PROGRAM MAIN
VAR_OUTPUT //globally readable, but only modifiable by MAIN
	outputBuffer : ARRAY[Surface.LEFT..Surface.RIGHT] OF Bundle;
	outputBufferPass, outputBufferFail : Bundle;
	numOutputBundles : USINT := 0;
	
	bundleIn : Bundle;
	bundleOut : Bundle;
	
	ready : BOOL;
	busy : BOOL;
	done : BOOL;
	error : BOOL;
	backlog : BOOL;
	
	localTime : TIMESTRUCT;
	pause : BOOL;
END_VAR
VAR
	removeBundle AT %I* : ARRAY[Surface.LEFT..Surface.RIGHT] OF BOOL;
	clearPassBuffer, clearFailBuffer AT %I* : BOOL;
	receiverStruct : AdsData;
	
	//ETA is not strictly required, area will process bundle even if it is not in ETA arrays
	expectedBundles : ARRAY[0..GVL.maxQueue] OF STRING; //bundles expected to arrive
	expectedArrivals : ARRAY[0..GVL.maxQueue] OF TIMESTRUCT; //bundles expected to arrive
	numEtaBundles : INT;
	
	//parallel arrays - bundle, bypass
	numBundlesQueue : INT;
	bundlesQueue : ARRAY[0..GVL.maxQueue] OF Bundle;
	bundlesBypass : ARRAY[0..GVL.maxQueue] OF BOOL;
	
	//spacerRecollector : PackagerFreeAsync;
	paperSection : PaperEx;
	cardboardCornerGuardSection : CardboardCornerGuardEx;
	chipboardSection : ChipboardEx;
	woodBunkSection : WoodBunkEx;
	outputSection : AreaOutputEx;
	run : ARRAY[0..SectionEnum.size] OF BOOL := [6(TRUE)];
	
	fbLocalSystemTime : FB_LocalSystemTime;
	fbEventLogger : SqlDatabaseAccessor;
	
	start : BOOL;
	
	processingMode : (PARALLEL, SINGLE, SERIAL, CLEAR);
	requestedMode : (PARALLEL, SINGLE, SERIAL, CLEAR);
	serialSection : REFERENCE TO SectionEx;
END_VAR
VAR //these variables are only tracked for HMI
	sectionsBusy : ARRAY[0..SectionEnum.size] OF BOOL;
	sectionsIterator : ARRAY[0..SectionEnum.size] OF INT;
END_VAR
VAR CONSTANT
	numSections : INT := 6;
	maxOutputBundles : USINT := 3;
END_VAR

demoHMI();

SizeCheck();
getLocalTime();

AdsClient( //PLC-PLC comms
	ServerNetId:= , 
	ServerPort:= , 
	bBusy=> , 
	err=> , 
	errid=> , 
	localPrgName=> , 
	localNetId=> , 
	localPort=> , 
	socketReady=> , 
	remoteAccessPrefix=> );
	
TcpServer1Vision( //PLC-Vision comms
	ServerNetId:= , 
	ServerAdr:= , 
	ServerPort:= , 
	busy=> , 
	error=> , 
	errorId=> , 
	bytesReceived=> , 
	connected=> , 
	receiveStruct=> );
	
IF NOT ( enableHardware() AND initialize() ) OR pause THEN
	RETURN;	
END_IF

//THIS MUST BE CALLED FIRST
CallHardware();
ConveyorControl();

IF AdsClient.fetchData(receiverStruct) THEN
	interpretTransmission(receiverStruct);
END_IF


IF ready AND BundleIsValid(bundleIn) THEN
	receive();
END_IF


IF NOT busy THEN
	processingMode := requestedMode;
END_IF
requestMode();

IF clearPassBuffer OR clearFailBuffer THEN
	transfer();
	shiftBundles();
END_IF

ready := paperSection.ready; //if A2 is not ready, dispatch controller must block operator from sending bundles here
busy := paperSection.busy OR cardboardCornerGuardSection.busy OR chipboardSection.busy OR woodBunkSection.busy OR outputSection.busy;
done := outputSection.done;
backlog := numBundlesQueue > 5;



fbEventLogger();

METHOD demoHMI : BOOL
VAR
	i : INT;
END_VAR
IF NOT start THEN //for HMI testing only, remove for production
	FOR i:=0 TO GVL.maxQueue BY 1 DO
		bundlesQueue[i].id := TO_STRING(i);
	END_FOR
	
	start := TRUE;
END_IF
END_METHOD

METHOD PRIVATE enableHardware : BOOL
VAR
	iCardboardSlot : CornerGuard := 1;
	iCornerGuardSlot : Cardboard := 1;
	iChipboardSlot : Chipboard := 1;
	iWoodBunkSlot : WoodBunk := 1;
	
	slotsArr : ARRAY[1..GVL.maxQueue] OF STRING;
	
	i : INT;
END_VAR
FOR iCardboardSlot:=1 TO Cardboard.size-1 BY 1 DO
	slotsArr[iCardboardSlot] := TO_STRING(iCardboardSlot);
END_FOR
cardboardSkidLeft.setupSlots(slotsArr);
cardboardSkidRight.setupSlots(slotsArr);


FOR iCornerGuardSlot:=1 TO CornerGuard.size-1 BY 1 DO
	slotsArr[iCornerGuardSlot] := TO_STRING(iCornerGuardSlot);
END_FOR
cornerGuardMagazineLeft.setupSlots(slotsArr);
cornerGuardMagazineRight.setupSlots(slotsArr);


FOR iChipboardSlot:=1 TO Chipboard.size-1 BY 1 DO
	slotsArr[iChipboardSlot] := TO_STRING(iChipboardSlot);
END_FOR
chipboardSkidLeft.setupSlots(slotsArr);
chipboardSkidRight.setupSlots(slotsArr);


FOR iWoodBunkSlot:=1 TO WoodBunk.size-1 BY 1 DO
	slotsArr[iWoodBunkSlot] := TO_STRING(iWoodBunkSlot);
END_FOR
woodBunkMagazineLeft.setupSlots(slotsArr);
woodBunkMagazineRight.setupSlots(slotsArr);


insertionA22Left.enable := TRUE;
insertionA21Left.enable := TRUE;

enableHardware := TRUE;
END_METHOD

METHOD PRIVATE getLocalTime : BOOL
fbLocalSystemTime(
	sNetID:= '', 
	bEnable:= TRUE, 
	dwCycle:= , 
	dwOpt:= , 
	tTimeout:= , 
	bValid=> , 
	systemTime=> localTime, 
	tzID=> );
	
getLocalTime := TRUE;
END_METHOD

METHOD PRIVATE initialize : BOOL
VAR
	i : INT;
	temp : POINTER TO BOOL;
END_VAR
paperSection.connectTo(ADR(cardboardCornerGuardSection));
cardboardCornerGuardSection.connectTo(ADR(chipboardSection));
chipboardSection.connectTo(ADR(woodBunkSection));
woodBunkSection.connectTo(ADR(outputSection));

paperSection.sectionID := SectionEnum.PAPER;
cardboardCornerGuardSection.sectionID := SectionEnum.CARDBOARD_CORNERGUARD;
chipboardSection.sectionID := SectionEnum.CHIPBOARD;
woodBunkSection.sectionID := SectionEnum.WOOD_BUNK;
outputSection.sectionID := SectionEnum.OUTPUT;

(*
	paperSection.accessNextSection := ADR(cardboardCornerGuardSection);
	cardboardCornerGuardSection.accessNextSection := ADR(chipboardSection);
	chipboardSection.accessNextSection := ADR(woodBunkSection);
	woodBunkSection.accessNextSection := ADR(outputSection);
	outputSection.accessNextSection := 0;
	
	outputSection.accessPrevSection := woodBunkSection;
	woodBunkSection.accessPrevSection := chipboardSection;
	chipboardSection.accessPrevSection := cardboardCornerGuardSection;
	cardboardCornerGuardSection.accessPrevSection := paperSection;
	paperSection.accessPrevSection := 0;
*)

(*
	12, 20	entry + paper
	9, 11	cardboard + corner guard
	5, 8	chipboard + wood bunk
	1, 4 	output buffer
	
	0, 0 	spacer recollector (possibly obsolete)
*)
ForceSetLifterConveyors();

paperSection.assignConveyors(12, 20);
cardboardCornerGuardSection.assignConveyors(9, 11);
chipboardSection.assignConveyors(5, 8);
woodBunkSection.assignConveyors(5, 8);
outputSection.assignConveyors(1, 4);

initialize := TRUE;
END_METHOD

METHOD PRIVATE interpretTransmission : BOOL
VAR_INPUT
	data : REFERENCE TO AdsData;
END_VAR
VAR
	i : INT;
END_VAR
CASE data.description OF
	EventsEnum.BUNDLE_IN:
		MEMCPY(ADR(bundleIn), ADR(data.binaryData), SIZEOF(bundleIn));
			
	EventsEnum.BUNDLE_ETA:
		MEMCPY(ADR(expectedBundles[numEtaBundles]), ADR(data.binaryData), SIZEOF(expectedBundles[numEtaBundles]));
		expectedArrivals[numEtaBundles] := data.timestamp;
		
END_CASE
END_METHOD

METHOD PRIVATE process : BOOL
(*
full parallel processsing
all sections may operate concurrently on any bundle
*)
paperSection(
	enable:= run[SectionEnum.PAPER], 
	bundlesQueue:= bundlesQueue, 
	bundlesBypass:= bundlesBypass,
	bundleOut=> , 
	bypass=> , 
	ready=> , 
	busy=> sectionsBusy[SectionEnum.PAPER], 
	done=> , 
	error=> , 
	backlog=> ,
	iBundle=> sectionsIterator[SectionEnum.PAPER],
	iPair=> );
	
cardboardCornerGuardSection(
	enable:= run[SectionEnum.CARDBOARD_CORNERGUARD],
	bundlesQueue:= bundlesQueue, 
	bundlesBypass:= bundlesBypass,
	bundleOut=> ,
	bypass=> , 
	ready=> , 
	busy=> sectionsBusy[SectionEnum.CARDBOARD_CORNERGUARD], 
	done=> , 
	error=> , 
	backlog=> ,
	iBundle=> sectionsIterator[SectionEnum.CARDBOARD_CORNERGUARD],
	iPair=> );

chipboardSection(
	enable:= run[SectionEnum.CHIPBOARD],
	bundlesQueue:= bundlesQueue, 
	bundlesBypass:= bundlesBypass, 
	bundleOut=> ,
	bypass=> , 
	ready=> , 
	busy=> sectionsBusy[SectionEnum.CHIPBOARD], 
	done=> , 
	error=> , 
	backlog=> ,
	iBundle=> sectionsIterator[SectionEnum.CHIPBOARD],
	iPair=> );

woodBunkSection(
	enable:= run[SectionEnum.WOOD_BUNK],
	bundlesQueue:= bundlesQueue, 
	bundlesBypass:= bundlesBypass, 
	bundleOut=> ,
	bypass=> , 
	ready=> , 
	busy=> sectionsBusy[SectionEnum.WOOD_BUNK], 
	done=> , 
	error=> , 
	backlog=> ,
	iBundle=> sectionsIterator[SectionEnum.WOOD_BUNK],
	iPair=> );
	
outputSection(
	enable:= run[SectionEnum.OUTPUT],
	bundlesQueue:= bundlesQueue, 
	bundlesBypass:= bundlesBypass,
	outputBuffer:= outputBuffer,
	bundleOut=> , 
	bypass=> , 
	ready=> , 
	busy=> sectionsBusy[SectionEnum.OUTPUT],
	done=> , 
	error=> , 
	backlog=> ,
	iBundle=> sectionsIterator[SectionEnum.OUTPUT],
	iPair=> );
END_METHOD

{attribute 'TcRpcEnable'}
METHOD PRIVATE receive : BOOL
VAR
	i : INT;
	shiftIndex : INT := -1;
	invalidBundle : Bundle;
END_VAR
FOR i:=0 TO GVL.maxQueue BY 1 DO //find the bundle in the ETA queue
	IF expectedBundles[i] = bundleIn.id THEN
		shiftIndex := i;
		EXIT;
	END_IF
END_FOR

IF shiftIndex > -1 THEN //if the bundle is found in the ETA queue, shift everything down
	MEMMOVE(
		ADR(expectedBundles[shiftIndex]), 
		ADR(expectedBundles[shiftIndex + 1]), 
		SIZEOF(STRING) * TO_UINT(GVL.maxQueue - shiftIndex));
		
	MEMMOVE(
		ADR(expectedArrivals[shiftIndex]), 
		ADR(expectedArrivals[shiftIndex + 1]), 
		SIZEOF(TIMESTRUCT) * TO_UINT(GVL.maxQueue - shiftIndex) );
		
	numEtaBundles := numEtaBundles - 1;
END_IF

FOR i:=0 TO GVL.maxQueue BY 1 DO
	IF BundleIsValid(bundlesQueue[i]) AND NOT bundlesBypass[i] THEN
		bundlesQueue[i] := bundleIn;
		bundlesBypass[i] := FALSE;
		
		receive := TRUE;
		RETURN;
	END_IF
END_FOR

IF NOT receive THEN
	error := TRUE;
END_IF
END_METHOD

METHOD requestMode : BOOL
CASE requestedMode OF
	PARALLEL:
		//backlog := numBundlesQueue >= 5;
		
	SINGLE:
		backlog := numBundlesQueue >= 1;
		
	SERIAL:
		backlog := numBundlesQueue >= 1;
		
	CLEAR:
		backlog := numBundlesQueue > 0;
		
END_CASE

CASE processingMode OF //run stations
	PARALLEL:
		process();
		backlog := numBundlesQueue >= 5;
		
	SINGLE:
		singleProcess();
		backlog := numBundlesQueue >= 1;
		
	SERIAL:
		serialProcess();
		backlog := numBundlesQueue >= 1;
		
	CLEAR:
		backlog := numBundlesQueue > 0;
		//stop processing
		
END_CASE
END_METHOD

METHOD serialProcess : BOOL
VAR_INPUT
END_VAR
(*
sections process bundles 1 by 1 in order
only 1 bundle allowed in the section at a time
*)
IF NOT __ISVALIDREF(serialSection) THEN
	serialSection REF= PaperSection;
END_IF

serialSection(
	enable:= TRUE, 
	sectionID:= , 
	bundlesQueue:= bundlesQueue, 
	bundlesBypass:= bundlesBypass, 
	bundleOut=> , 
	bypass=> , 
	ready=> , 
	busy=> , 
	done=> , 
	error=> , 
	backlog=> , 
	iBundle=> , 
	iPair=> );
	
IF serialSection.done THEN
	serialSection REF= serialSection.accessNextSection^;
END_IF
END_METHOD

METHOD shiftBundles : BOOL
VAR_INPUT
END_VAR
//shift down parallel arrays
MEMMOVE(ADR(bundlesQueue[0]), ADR(bundlesQueue[1]), SIZEOF(Bundle) * TO_UINT(GVL.maxQueue));
MEMMOVE(ADR(bundlesBypass[0]), ADR(bundlesBypass[1]), SIZEOF(BOOL) * TO_UINT(GVL.maxQueue));

//decrement each section's iterator to realign with their correct bundle
paperSection.shiftIterator();
cardboardCornerGuardSection.shiftIterator();
chipboardSection.shiftIterator();
woodBunkSection.shiftIterator();
outputSection.shiftIterator();
END_METHOD

METHOD singleProcess : BOOL
VAR_INPUT
END_VAR
(*
all sections may operate on a bundle as they arrive
only 1 bundle may enter the area at a time
*)
END_METHOD

METHOD PRIVATE transfer : BOOL
VAR
	i : INT;
END_VAR
//send TCP/ADS transmission back to Dispatch once bundle is removed from the plant

IF clearPassBuffer THEN
	fbEventLogger.queueEvent(event:= EventsEnum.BUNDLE_OUT); //modify to include bundle ID
	outputBufferPass := GVL.nullBundle;
END_IF

IF clearFailBuffer THEN
	fbEventLogger.queueEvent(event:= EventsEnum.BUNDLE_OUT); //modify to include bundle ID
	outputBufferFail := GVL.nullBundle;
END_IF
END_METHOD

END_PROGRAM

(* stored: Version 1.1.0.1, ProductVersion 3.1.4024.11
   POU MAIN: Id {f8ea2e52-8cdd-4c5a-a5f9-4c8d8a3c6a2c}, SpecialFunc None
   Folder Process Modes: Id {8d1d624d-f207-4b80-ae71-4f41b10197eb}
   Folder Setup: Id {766689c6-4b05-4d8b-a8a4-3bf5c2750aa3}
   Method demoHMI: Id {73fc04c3-3b20-4b90-b668-e45a325d9c2c}
   Method enableHardware: Id {0ba728b9-6522-4c82-81e3-44efce8fc95c}
   Method getLocalTime: Id {b9dfd14b-062f-4ab4-b051-cd1816451bba}
   Method initialize: Id {1af4c629-041d-43ca-9e16-2266f17c58c8}
   Method interpretTransmission: Id {04aa253b-ab0d-41b0-b6b2-443fd8efedd5}
   Method process: Id {f9da02b9-c065-4582-840f-d291dad1e576}
   Method receive: Id {2de20b6b-9727-4ca1-a75e-22c752a3c085}
   Method requestMode: Id {64bfef98-63a1-42bb-a7e6-1c650a0eba17}
   Method serialProcess: Id {47421198-a334-44b3-b4bd-005760b5320c}
   Method shiftBundles: Id {5473c570-b523-4be9-bf64-c8f58c1af44e}
   Method singleProcess: Id {61419f9a-4fd7-4611-81f5-1ecc6e826cfd}
   Method transfer: Id {a55e1076-0c29-4969-952a-05c194ea9e2d} *)
